PROGRAM POU_PLUS
VAR
	Result:REAL;
	Value01:REAL;
	Value02:REAL;
	
END_VAR

Result:=Value01+Value02;

END_PROGRAM

(* stored: Version 1.1.0.1, ProductVersion 3.1.4024.4
   POU POU_PLUS: Id {a9e91d33-6a20-4b41-8e72-7456877034a3}, SpecialFunc None *)
